{attribute 'qualified_only'}
VAR_GLOBAL
	fbEventTrigger : FB_EventTrigger(TC_EVENT_CLASSES.TestEventClass); 
END_VAR

(* stored: Version 1.1.0.1, ProductVersion 3.1.4026.13
   GVL GVL_Fault: Id {65ce6d33-01de-4307-8203-70a1f3546c49} *)
